FUNCTION f_Multiplication : REAL
VAR_INPUT
	rProd1	:	REAL;
	rProd2	:	REAL;
END_VAR
VAR
END_VAR

f_Multiplication := rProd1	* rProd2;

END_FUNCTION

(* stored: Version 1.1.0.1, ProductVersion 3.1.4024.12
   POU f_Multiplication: Id {b7cc7ed1-b28d-4040-9aa5-4dd3a2646a27}, SpecialFunc None *)
